PROGRAM PRG_FB_UpsCx20xx_Test
VAR
	iSample		: INT := 10;
	fbUpsCX2020	: FB_UpsCx2xxx;
END_VAR

VAR PERSISTENT
	iSamplePersistent : INT := 10;
END_VAR

fbUpsCX2020.MR_FirstCycle( sName := 'Beckhoff UPS CX2020',
							sNetID := '',
							iPlcPort := 852,
							tTimeout := DEFAULT_ADS_TIMEOUT);

fbUpsCX2020();

END_PROGRAM

(* stored: Version 1.1.0.1, ProductVersion 3.1.4024.9
   POU PRG_FB_UpsCx20xx_Test: Id {358a48eb-c17b-4047-939c-9eda2716e834}, SpecialFunc None *)
